PROGRAM P_Rum_5_341
VAR
//Light

	fbLys		: FB_Light_Type_A;
	
	stDaliSetup	: SH_Light.ST_DALI_RoomSetup := (		byShrtAdr_Prim := 5, 
														byGrpAdr_Prim := 2, 
														eMod_Prim := E_DALIAddressType.Group, 
														byShrtAdr_Sec := 1, 
														byGrpAdr_Sec := 1, 
														eMod_Sec := E_DALIAddressType.Short, 
														byShrtAdr_Supl := 1, 
														DALI_LINE_NUM_PRIM := DALI_LINE_NUM_LIGHT, 
														DALI_LINE_NUM_SEC := 0, //0 = ingen zonestyring/vinduerække
														DALI_LINE_NUM_SUPL := DALI_LINE_NUM_PENDANTS);
	stLiveData				: SH_Light.ST_LiveData;
	//stLiveData AT %MB22	: SH_Light.ST_LiveData;
	bTopButtonZone1			: BOOL;
	bTopButtonZone1_Visu	: BOOL;
	bBottomButtonZone1		: BOOL;
	bBottomButtonZone1_Visu	: BOOL;
	bButtonZone2			: BOOL;
	fLuxOn					: REAL := 500;
	fLuxDim					: REAL := 200;
	tPIRDim					: TIME := T#15M;
	tPIROff					: TIME := T#30M;
	fOffsetSec				: REAL := 20;
	bOccupiedRoom			: BOOL;

	bRunTuning				: BOOL;
	
// Sensor Settings
	fbSensor					: SH_Light.FB_NIKO_P46xx_1Pcs;
	//fbSensor					: SH_Light.FB_NIKO_P46xx_2Pcs;
	bySensorAddr				: BYTE := 2;
	//arrSensorAddr				: ARRAY[1..2] OF BYTE := [9,10];
	bInitialize					: BOOL := TRUE;
	stDaliSensorSetup			: ST_DALI_NIKOP46SetupData;
	bInitErr					: BOOL;
	bInitDone					: BOOL;
	//arrInitErr					: ARRAY [1..2] OF BOOL;
	//arrInitDone					: ARRAY [1..2] OF BOOL;
	arrSensorScales				: ARRAY [1..10] OF SH_Light.ST_DALI_SensorScaleMode := [	(fMeassureMaxSensor := 1023, fReadMaxSensor := 1023),
																						9(())];
	bCancelHoldTimerOccupancy	: BOOL;
(*	eEventPriorityOccupancy		: E_DALIEventPriority := E_DALIEVENTPRIORITY.Middle;
	nHoldTimerOccupancy			: WORD := 5; // Value in s. 	
	nReportTimerOccupancy		: BYTE := 120; // Value in s, Preset manufacturer value
	nDeadtimeTimerOccupancy		: WORD := 100; // Value in ms, Predefined Value of DALI Standard
	bCancelHoldTimerOccupancy	: BOOL;
	nSensitivityOccupancy		: BYTE:= 3; //setting Sensivity (0..4) 0 (Off), 1 (Min), 2(Low), 3(High) and 4 (Max)

	bEnableLuxEvent				: BOOL;
	eEventPriorityBrightness	: E_DALIEventPriority := E_DALIEVENTPRIORITY.Middle;
	nDeadtimeTimerBrightness	: WORD := 1500; // Value in ms, Predefined Value of DALI Standard
	nHysteresisBrightness		: BYTE := 2; // Value in %
	nHysteresisMinBrightness	: BYTE := 10; // Absolute Value, depending on the manufacturer specific resolution
	nReportTimerBrightness		: BYTE := 120; // Value in s, Preset manufacturer value
*)

END_VAR

VAR CONSTANT
	Sensor_DALI_LINE_NUM	: BYTE := 2;
	DALI_LINE_NUM_LIGHT		: BYTE := 1;
	DALI_LINE_NUM_PENDANTS	: BYTE := 0; //0=ingen pendler
END_VAR
VAR PERSISTENT
	stPirSensorData: SH_Light.ST_DALI_Sensor;
	stTuneData: SH_Light.ST_TuneData_EX;
END_VAR

A_Buttons();
A_LightCtrl();
A_Sensor();

ACTION A_Buttons:
bTopButtonZone1		:= GVL_EnOcean.strEnOceanSwitch_Rum_5_341.bT1_ON OR bTopButtonZone1_Visu;
bBottomButtonZone1	:= GVL_EnOcean.strEnOceanSwitch_Rum_5_341.bT1_OFF OR bBottomButtonZone1_Visu;
END_ACTION

ACTION A_LightCtrl:

fbLys(
	nZoneID:= 1, 
	bButtonZone1:= bTopButtonZone1,
	bBottomButtonZone1 := bBottomButtonZone1, 
	bButtonZone2:= bButtonZone2, 
	fLuxOn:= fLuxOn, 
	fLuxDim:= fLuxDim, 
	tPIRDim:= tPIRDim, 
	tPIROff:= tPIROff, 
	fOffsetSec:= fOffsetSec, 
	bReInit:= , 
	stDaliSetup:= stDaliSetup, 
	ipCommunication_Prim:= P_DALI_Background.arrfbKL6821Communication[DALI_LINE_NUM_LIGHT], 
	ipCommunication_Sec:= P_DALI_Background.arrfbKL6821Communication[DALI_LINE_NUM_LIGHT], 
	ipCommunication_Supl:= P_DALI_Background.arrfbKL6821Communication[DALI_LINE_NUM_LIGHT], 
	fMinOutputPowerLevelRoom:= 15, 
	fMaxOutputPowerLevelRoom:= 100, 
	nCycleTimeInMS:= 10 , 
	bRunTuning:= bRunTuning, 
	bOccupiedRoom=> bOccupiedRoom, 
	bError_Prim=> , 
	nError_Prim=> , 
	stTuneData:=stTuneData , 
	stPirSensorData:= stPirSensorData, 
	stLiveData:= stLiveData);
END_ACTION

ACTION A_Sensor:

fbSensor.ipCommunication := P_DALI_Background.arrfbKL6821Communication[Sensor_DALI_LINE_NUM];


fbSensor(
	byShrtAdr:= bySensorAddr,
	bInitialize:= bInitialize, 
	DALI_LINE_NUM:= Sensor_DALI_LINE_NUM, 
 	//bCancelHoldTimerOccupancy:= bCancelHoldTimerOccupancy, 
	stSensorSetup := stDaliSensorSetup,
	bInitErr=> bInitErr, 
	bInitDone=> bInitDone,
	stPirSensorData:= stPirSensorData, 
	arrSensorScales:= arrSensorScales);

(*
fbSensor(
	arrShrtAdr:= arrSensorAddr,
	bInitialize:= bInitialize, 
	DALI_LINE_NUM:= Sensor_DALI_LINE_NUM, 
 	//bCancelHoldTimerOccupancy:= bCancelHoldTimerOccupancy, 
	stSensorSetup := stDaliSensorSetup,
	arrInitErr=> arrInitErr, 
	arrInitDone=> arrInitDone,
	stPirSensorData:= stPirSensorData, 
	arrSensorScales:= arrSensorScales);
	*)
END_ACTION

END_PROGRAM

(* stored: Version 1.1.0.1
   POU P_Rum_5_341: Id {a7b61f30-4143-4bcb-b26f-268a479d30ef}, SpecialFunc None
   Action A_Buttons: Id {3d2cd758-973c-48ea-995b-d0eadb41d008}
   Action A_LightCtrl: Id {45d3efd6-6f1b-4cbf-a25f-825ad301bb77}
   Action A_Sensor: Id {78695773-a4f3-46f0-bb76-57645ea4add1} *)
